FUNCTION_BLOCK X2Y2I (* Compute X^2-Y^2(INT) *)
  (* Standard: 61499-1 *)
  (* Version 0.1, 2004-06-07, JHC, HUT *)
  (* Version 0.0, 2003-08-17, JHC, Rockwell Automation, Adapted from X2Y2. *)
  (* Compiler header: package fb.rt.student; import fb.rt.plc.math.*; *)
  (* Compiler Java IBM Jikes 1.0.6 *)
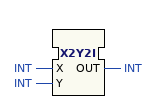
  VAR_INPUT
    X : INT;
    Y : INT;
  END_VAR
  VAR_OUTPUT
    OUT : INT;
  END_VAR
  ALGORITHM REQ IN FBD: (* Normally executed algorithm *)
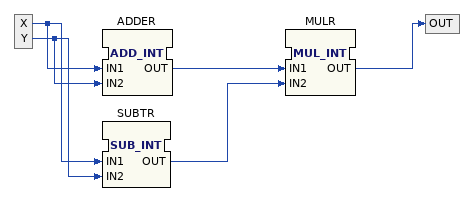
    FBS
      ADDER : ADD_INT;
      SUBTR : SUB_INT;
      MULR : MUL_INT;
    END_FBS
    DATA_CONNECTIONS
      X TO ADDER.IN1;
      Y TO ADDER.IN2;
      X TO SUBTR.IN1;
      Y TO SUBTR.IN2;
      ADDER.OUT TO MULR.IN1;
      SUBTR.OUT TO MULR.IN2;
      MULR.OUT TO OUT;
    END_CONNECTIONS
  END_ALGORITHM
END_FUNCTION_BLOCK
